//==================================================================================================
//							Beckhoff Automation Poland
//									11.04.2018
//	This object shall provide the text id of the last DiagMessage of type error, which occurred in this axis.
//  v1.0	|| TC v 3.1.4022.16		|| - pierwsza wersja
//==================================================================================================
FUNCTION_BLOCK FB_ReadChannelErrorCodeAX8000_1
VAR_INPUT
	bExecute 						: BOOL;
	stDriveRef						: ST_DriveRef;						// 
END_VAR
VAR_OUTPUT
	bBusy							: BOOL;
	bError							: BOOL; 							// General error: parameter or CoE read.
	iAdsErrId						: UINT;								// Forwarded output FB_CoERead_ByDriveRef
	iCANopenErrId					: UINT;								// Forwarded output FB_CoERead_ByDriveRef
	uiChannelErrorCode				: UINT;								// 603F Error code	0x603F (Ch A)/ 0x683F (Ch B) 	UINT16
	{attribute 'displaymode':='hex'}
	uiChannelErrorCodeHex			: UINT;								// 603F Error code	0x603F (Ch A)/ 0x683F (Ch B) 	UINT16
END_VAR
VAR
	fbCoERead						: FB_CoERead_ByDriveRef;			// FB for read CoE parameters
END_VAR

fbCoERead(	stDriveRef					:= stDriveRef,
			nIndex						:= 16#603F + (stDriveRef.nDriveNo * 16#800),
			nSubIndex					:= 0,
			pDstBuf						:= ADR(uiChannelErrorCode),
			cbBufLen					:= SIZEOF(uiChannelErrorCode),
			bExecute					:= bExecute,
			bBusy						=> bBusy,
			bError						=> bError,
			iAdsErrId					=> iAdsErrId,
			iCANopenErrId				=> iCANopenErrId);

uiChannelErrorCodeHex					:= uiChannelErrorCode;

END_FUNCTION_BLOCK

(* stored: Version 1.2.0.0, ProductVersion 3.1.4026.13, FileIdentifier 210be905d23e5d27d35118ff1fa38912900af974, FileSignature 165b83699d7d13f27ffa8c4175e061305a0414259a4d1449da69dce2b7f57d1956827f4e24e3219a86dbde78009581765c4865921fe64d4720001a805891c28fc20cb9ba5c40cfcd2aabb5ef68b32dfabca38ff4509d6bb2e0526bd4649390358dbb51e8540e41806a53baf9a7e51f9e917948087aa4ecb65efdb78d3532b4e3dcd83ea7f1c4f79276cfabc8d8ee82f762c1a65d0ba7d26b48a0a4985c96afb729d6dd0839f3bcd77abdbf3f6b442ccb70811fe0099cfb2c5d6cb93b92f7aeea4d84c5bdeadce7a81519e06fffe24a11245748373eb03ddca0a3934a52cf451be856092081bda745b55803875fae76e32b4fbe9417d1898ba266c41c2394af59
   POU FB_ReadChannelErrorCodeAX8000_1: Id {0aa7b657-a1e3-47ea-9de3-c0add7bdb88c}, SpecialFunc None *)
